(* Logix 5000 project; controller EuniceF_ICA18 vendor 1 type 14 code 150 rev 37.11; software revision 37.00 *)

TASK MainTask (continuous, watchdog 500 ms) : MainProgram

MODULES
   Local : vendor 1 type 14 code 150 (Compact 0, rev 37.11)
      Discrete_IO : Embedded (Compact 1, rev 3.1, Output RPI 20 ms)
      Analog_IO : Embedded (Compact 2, rev 1.1, Output RPI 80 ms)
      Counters : Embedded (Compact 3, rev 1.1, Output RPI 20 ms)
END_MODULES

VAR_GLOBAL   (* controller tags *)
   East_Amber : ALIAS FOR Local:1:O.Data.6;
   East_Green : ALIAS FOR Local:1:O.Data.7;
   East_Red : ALIAS FOR Local:1:O.Data.5;
   East_Wapper : ALIAS FOR Local:1:O.Data.15;
   North_Amber : ALIAS FOR Local:1:O.Data.2;
   North_Green : ALIAS FOR Local:1:O.Data.3;
   North_Red : ALIAS FOR Local:1:O.Data.1;
   SEQ : DINT;
   StateEWAmber : DINT := 1;
   StateEWGreen : DINT;
   StateNSAmber : DINT;
   StateNSGreen : DINT;
   StatusEW : STRING;
   StatusNS : STRING;
   StrAmber : STRING := 'Amber';
   StrGreen : STRING := 'Green';
   StrLight : STRING := 'Light : ';
   StrRed : STRING := 'Red';
   Timer2s : TIMER := (PRE := 2000);
   Timer4s : TIMER := (PRE := 4000);
   Timer6s : TIMER := (PRE := 6000);
END_VAR

PROGRAM MainProgram   (* main routine MainRoutine *)

ROUTINE MainRoutine   (* ladder *)
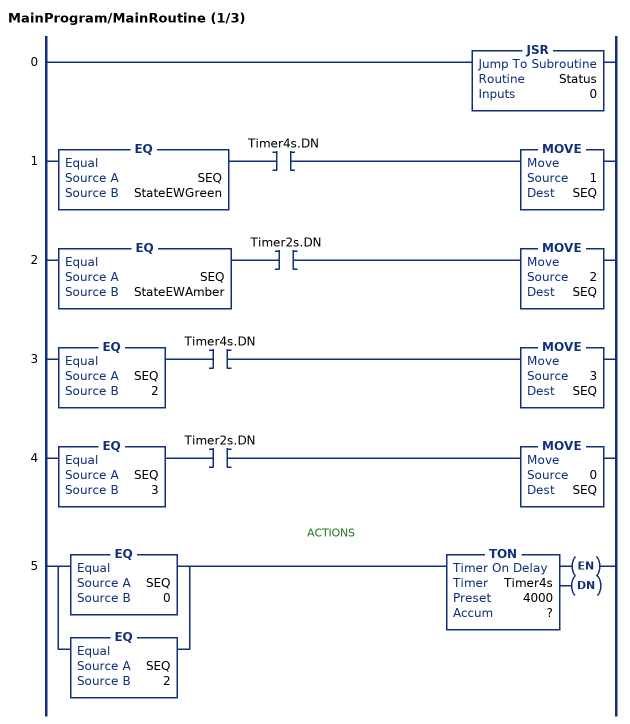
   0: JSR(Status,0);
   1: EQ(SEQ,StateEWGreen)XIC(Timer4s.DN)MOVE(1,SEQ);
   2: EQ(SEQ,StateEWAmber)XIC(Timer2s.DN)MOVE(2,SEQ);
   3: EQ(SEQ,2)XIC(Timer4s.DN)MOVE(3,SEQ);
   4: EQ(SEQ,3)XIC(Timer2s.DN)MOVE(0,SEQ);
   // ACTIONS
   5: [EQ(SEQ,0) ,EQ(SEQ,2) ]TON(Timer4s,?,?);
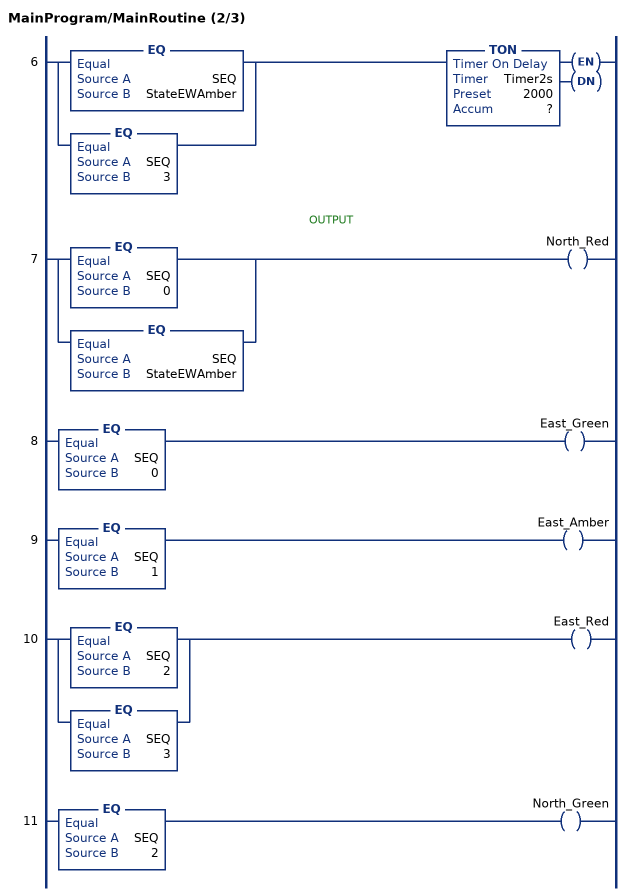
   6: [EQ(SEQ,StateEWAmber) ,EQ(SEQ,3) ]TON(Timer2s,?,?);
   // OUTPUT
   7: [EQ(SEQ,0) ,EQ(SEQ,StateEWAmber) ]OTE(North_Red);
   8: EQ(SEQ,0)OTE(East_Green);
   9: EQ(SEQ,1)OTE(East_Amber);
   10: [EQ(SEQ,2) ,EQ(SEQ,3) ]OTE(East_Red);
   11: EQ(SEQ,2)OTE(North_Green);
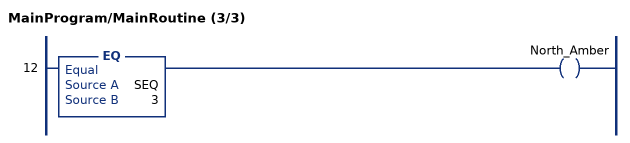
   12: EQ(SEQ,3)OTE(North_Amber);
END_ROUTINE

ROUTINE Status   (* structured text *)
   if SEQ = StateEWGreen then
   
   	concat(StrLight, StrGreen, StatusEW);
   	concat(StrLight, StrRed, StatusNS);
   
   end_if;
   
   if SEQ = StateEWAmber then
   
   	concat(StrLight, StrAmber, StatusEW);
   	concat(StrLight, StrRed, StatusNS);
   
   end_if;
   
END_ROUTINE
END_PROGRAM
